// TIA Portal V18 export
VAR_GLOBAL   // PLC tag table "S2_R1"
   S2_R1_Valve_Up AT %Q500.0 : Bool;
   S2_R1_Valve_Down AT %Q500.1 : Bool;
   S2_R1_Sen_Drv_1 AT %Q500.2 : Bool;
   S2_R1_Sen_Drv_2 AT %Q500.3 : Bool;
   S2_R1_Sen_Drv_3 AT %Q500.4 : Bool;
   S2_R1_Sen_Drv_4 AT %Q500.5 : Bool;
   S2_R1_Sen_Val1_Up AT %Q500.6 : Bool;
   S2_R1_Sen_Val1_Down AT %Q500.7 : Bool;
   S2_R1_Sen_Val2_Up AT %Q501.0 : Bool;
   S2_R1_Sen_Val2_Down AT %Q501.1 : Bool;
   S2_R1_Hyd_Filtr AT %Q501.2 : Bool;
   S2_R1_Hyd_Empty AT %Q501.3 : Bool;
   S2_R1_Safety1_1 AT %I550.0 : Bool;
   S2_R1_Safety2_1 AT %I550.1 : Bool;
   S2_R1_Safety3_1 AT %I550.2 : Bool;
   S2_R1_Safety4_1 AT %I550.3 : Bool;
   S2_R1_Safety1_2 AT %I550.4 : Bool;
   S2_R1_Safety2_2 AT %I550.5 : Bool;
   S2_R1_Safety3_2 AT %I550.6 : Bool;
   S2_R1_Safety4_2 AT %I550.7 : Bool;
END_VAR
